(****************************************************************************************)
(*							Beckhoff Automation Poland									*)
(*							L_TBSetBitOfByte v1.0										*)
(*									29.02.2007											*)
(*				This function sets a single bit in a value of type ”byte” to “1”		*)
(*______________________________________________________________________________________*)
FUNCTION L_TBSetBitOfByte : BYTE
VAR_INPUT
	byInput: BYTE;
	byBitNr: BYTE;
END_VAR

L_TBSetBitOfByte := byInput;
CASE byBitNr OF
	0:
	L_TBSetBitOfByte.0 := TRUE;
	1:
	L_TBSetBitOfByte.1 := TRUE;
	2:
	L_TBSetBitOfByte.2 := TRUE;
	3:
	L_TBSetBitOfByte.3 := TRUE;
	4:
	L_TBSetBitOfByte.4 := TRUE;
	5:
	L_TBSetBitOfByte.5 := TRUE;
	6:
	L_TBSetBitOfByte.6 := TRUE;
	7:
	L_TBSetBitOfByte.7 := TRUE;
END_CASE

END_FUNCTION

(* stored: Version 1.1.0.1, ProductVersion 3.1.4026.13, FileIdentifier 3b9779b281241499e70a569c7dfd11bbc3c36746, FileSignature 161cefb1d763fde4d45de7fc564bc46042906476d6fc20324d4d35bd21a7b4b95214ec8aa4e9f1fe02cbeed24d9c76ace6b254f8f2d9c8fd2990271cb3343e2dc56d09b9d408dc6b42d2d3a788500f4ef437473bb36847486c714976e0aff46f456deac286f28d3dca1abeef31455e207ab1b287ce9d39355c7f809db99c02c3e4729eea094a81e5d27d7246888543d1274e6a3bae0850907334df92cd0fc22dcbe00c3508f13e6f35b958034daab080426f76d3225fca47dd54a50445c8e32d83fcc50ff16addf672e6661ea7f519b04fcaaf98ecf34a352d92a432598092ea8d3f0e9b307e6c86b81aaea16a7c81ce18e5398ca1e1067f0c732ccb0cb5f45e
   POU L_TBSetBitOfByte: Id {29345edb-33a7-4130-bbe0-e906ef1a51bf}, SpecialFunc None *)
